{attribute 'GeneratedUsingTerminal: EK1100-0000-0018'}
{attribute addProperty BoxType "EK1100-0000-0018"}
{attribute addProperty Id "Beckhoff_EQ3xxxEK1122Beckhoff_EQ3xxxEK1122_D437BD35718"}
{attribute addProperty CRC "260553954"}
{attribute addProperty Size "718"}
TYPE Beckhoff_EQ3xxx_0F87BCE2 EXTENDS EK1100_1FC0878B :
STRUCT
	{attribute addProperty Name "Beckhoff_EQ3xxxEK1122"}
	Beckhoff_EQ3xxxEK1122 : Beckhoff_EQ3xxxEK1122_D437BD35;
END_STRUCT
END_TYPE

(* stored: Version 1.2.0.0, ProductVersion 3.1.4024.9
   DUT Beckhoff_EQ3xxx_0F87BCE2: Id {80353d79-ebbc-4b7b-8629-82d0ef095268} *)
